// TIA Portal V16 export
// export: Created 2021-07-12T14:47:07.8764682Z, ExportSetting WithDefaults, DisplayName Totally Integrated Automation Portal, DisplayVersion V16, DisplayName TIA Portal Version Control Interface, DisplayVersion V16, DisplayName TIA Portal Openness, DisplayVersion V16, DisplayName STEP 7 Professional, DisplayVersion V16, DisplayName STEP 7 Safety, DisplayVersion V16, DisplayName WinCC Professional, DisplayVersion V16
FUNCTION_BLOCK "SimaHydTO_AxisAdvanced_PosAxis"   // FB33111, FBD
TITLE = SimaHydTO_AxisAdvanced_PosAxis
{ S7_Optimized_Access := 'TRUE' }
FAMILY : SimaHydTO/LAxisBasics
VERSION : 1.0
// Function block information: See Function block network 1
// stored: AutoNumber true, IsIECCheckEnabled false, IsRetainMemResEnabled false, MemoryReserve 100, SetENOAutomatically false, UDAEnableTagReadback false
   VAR_INPUT
      axis : TO_PositioningAxis;   // Technology object (axis)
      moveRelativeExecute : Bool;   // MC_MoveRelative: Start job with a positive edge
      moveRelativeDistance : LReal := 0.0;   // Distance of relative movement
      moveAbsoluteExecute : Bool;   // MC_MoveAbsolute: Start job with a positive edge
      moveAbsolutePosition : LReal := 0.0;   // Target position of absolute movement
      moveAbsoluteDirection : Int := 1;   // Direction of absolute movement: 0: Positive direction / 1: Negative direction / 3: Shortest direction
      moveAbsPositionControlled : Bool := true;   // 0: Non position-controlled operation / 1: Position-controlled mode - The parameter applies as long as the MC_MoveJog command is executed. After this, the setting of MC_Power applies again.
      haltExecute : Bool;   // MC_Halt: Start job with a positive edge
      haltAbortAcceleration : Bool := false;   // Acceleration control: False: The current acceleration at the start of the job is reduced using the configured jerk. Afterwards, the deceleration builds up / True: The acceleration is set to 0.0 at the start of the job, and the deceleration immediately builds up.
      Velocity : LReal := 100.0;   // Velocity of movement
      Acceleration : LReal := -1.0;   // Acceleration of movement
      Deceleration : LReal := -1.0;   // Deceleration of movement
      Jerk : LReal := -1.0;   // Jerk of movement
   END_VAR
   VAR_OUTPUT
      moveRelativeDone { ExternalWritable := 'False'} : Bool;   // MC_MoveRelative: Job is completed
      moveRelativeBusy { ExternalWritable := 'False'} : Bool;   // MC_MoveRelative: Job is running
      moveAbsoluteDone { ExternalWritable := 'False'} : Bool;   // MC_MoveAbsolute: Job is completed
      moveAbsoluteBusy { ExternalWritable := 'False'} : Bool;   // MC_MoveAbsolute: Job is running
      haltDone { ExternalWritable := 'False'} : Bool;   // MC_Halt: Job is running
      haltBusy { ExternalWritable := 'False'} : Bool;   // MC_Halt: Job is running
      commandAborted { ExternalWritable := 'False'} : Bool;   // The job was aborted by another job during execution (see also StatusID)
      error { ExternalWritable := 'False'} : Bool;   // An error occurred during execution of the job. The job is rejected. The cause of the error can be found in the "ErrorID" parameter.
      errorID { ExternalWritable := 'False'} : Word;   // ErrorID of motion control instruction (see also StatusID)
      statusID { ExternalWritable := 'False'} : Int;   // Additional specification of affected Motion control instruction of CommandAborted or Error: 0: No instruction / 1: MC_MoveRelative / 2: MC_MoveAbsolute / 3: MC_Halt
   END_VAR
   VAR
      instMcMoveRelative { ExternalAccessible := 'False'; ExternalVisible := 'False'; ExternalWritable := 'False'; S7_SetPoint := 'True'} : MC_MOVERELATIVE;   // PLCopen functions of basic motion control
      instMcMoveAbsolute { ExternalAccessible := 'False'; ExternalVisible := 'False'; ExternalWritable := 'False'; S7_SetPoint := 'True'} : MC_MOVEABSOLUTE;
      instMcHalt { ExternalAccessible := 'False'; ExternalVisible := 'False'; ExternalWritable := 'False'; S7_SetPoint := 'True'} : MC_HALT;
      statCommandAborted { ExternalAccessible := 'False'; ExternalVisible := 'False'; ExternalWritable := 'False'} : Array[#ARRAY_BEGIN..#ARRAY_END] of Bool;   // Arrays to save error information of PLCopen functions
      statError { ExternalAccessible := 'False'; ExternalVisible := 'False'; ExternalWritable := 'False'} : Array[#ARRAY_BEGIN..#ARRAY_END] of Bool;
      statErrorID { ExternalAccessible := 'False'; ExternalVisible := 'False'; ExternalWritable := 'False'} : Array[#ARRAY_BEGIN..#ARRAY_END] of Word;
      instMoveAbsOpenLoop { S7_SetPoint := 'True'} : "LSimaHydTO_MC_MoveAbsOpenLoop";
   END_VAR
   VAR_TEMP
      tempDwordCommandAborted : DWord;   // Variables to check error informations of PLCopen functions
      tempDwordError : DWord;
      tempCount : Int;   // Counter of FOR counting loop
   END_VAR
   VAR CONSTANT
      ARRAY_BEGIN : Int := 1;   // Start-Index of array (Maximum 32 Array elements!)
      ARRAY_END : Int := 32;   // End-Index of array (Maximum 32 Array elements!)
      ERROR_DEFAULT : Bool := false;   // Default values of output signals
      ERRORID_DEFAULT : Word := 16#0;
      STATUSID_DEFAULT : Int := 0;
   END_VAR
BEGIN

REGION Network 1 (SCL): Axis Basics - Header
   //=============================================================================
   //SIEMENS AG
   //(c)Copyright 2016 All Rights Reserved
   //-----------------------------------------------------------------------------
   //Library:       AxisAdvanced
   //Tested with:   S7-1500 V2.5
   //Engineering:   TIA Portal V15
   //Restrictions:  Motion Control Library V4.0
   //Requirements:  S7-1500(T)
   //Functionality: Advanced axis control of TO_PositioningAxis
   //-----------------------------------------------------------------------------
   //Change log table:
   //Version  Date       Expert in charge Changes applied
   //01.00.00 19.07.2019 ArSc             First released version
   //=============================================================================
END_REGION

REGION Network 2: Axis Advanced - MC_MoveRelative
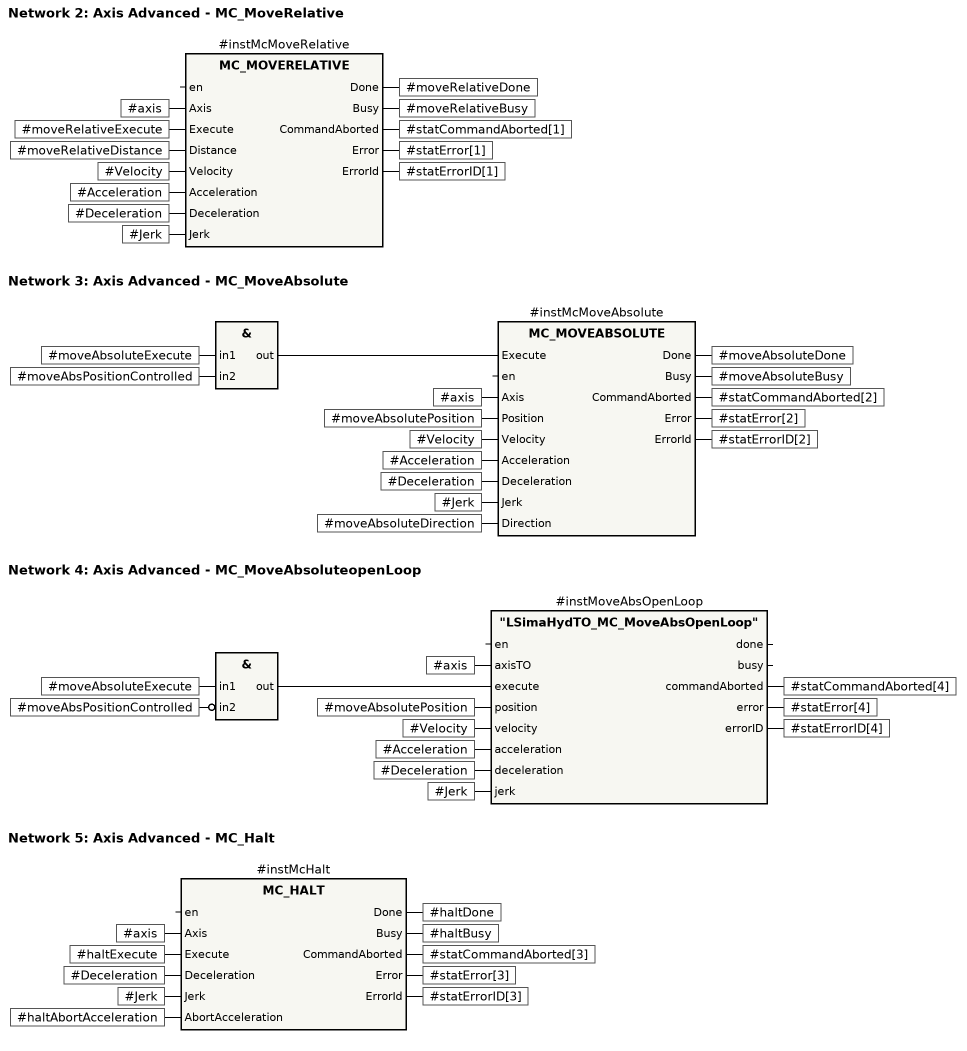
   #instMcMoveRelative(Axis := #axis,   // MC_MOVERELATIVE
                       Execute := #moveRelativeExecute,
                       Distance := #moveRelativeDistance,
                       Velocity := #Velocity,
                       Acceleration := #Acceleration,
                       Deceleration := #Deceleration,
                       Jerk := #Jerk,
                       Done => #moveRelativeDone,
                       Busy => #moveRelativeBusy,
                       CommandAborted => #statCommandAborted[1],
                       Error => #statError[1],
                       ErrorId => #statErrorID[1]);
END_REGION

REGION Network 3: Axis Advanced - MC_MoveAbsolute
   #instMcMoveAbsolute(Execute := #moveAbsoluteExecute AND #moveAbsPositionControlled,   // MC_MOVEABSOLUTE
                       Axis := #axis,
                       Position := #moveAbsolutePosition,
                       Velocity := #Velocity,
                       Acceleration := #Acceleration,
                       Deceleration := #Deceleration,
                       Jerk := #Jerk,
                       Direction := #moveAbsoluteDirection,
                       Done => #moveAbsoluteDone,
                       Busy => #moveAbsoluteBusy,
                       CommandAborted => #statCommandAborted[2],
                       Error => #statError[2],
                       ErrorId => #statErrorID[2]);
END_REGION

REGION Network 4: Axis Advanced - MC_MoveAbsoluteopenLoop
   #instMoveAbsOpenLoop(axisTO := #axis,   // "LSimaHydTO_MC_MoveAbsOpenLoop"
                        execute := #moveAbsoluteExecute AND NOT #moveAbsPositionControlled,
                        position := #moveAbsolutePosition,
                        velocity := #Velocity,
                        acceleration := #Acceleration,
                        deceleration := #Deceleration,
                        jerk := #Jerk,
                        commandAborted => #statCommandAborted[4],
                        error => #statError[4],
                        errorID => #statErrorID[4]);
END_REGION

REGION Network 5: Axis Advanced - MC_Halt
   #instMcHalt(Axis := #axis,   // MC_HALT
               Execute := #haltExecute,
               Deceleration := #Deceleration,
               Jerk := #Jerk,
               AbortAcceleration := #haltAbortAcceleration,
               Done => #haltDone,
               Busy => #haltBusy,
               CommandAborted => #statCommandAborted[3],
               Error => #statError[3],
               ErrorId => #statErrorID[3]);
END_REGION

REGION Network 6 (SCL): Axis Basics - Generate output signals and error detection
   //General output signals

   //Reset output signals
   #commandAborted := False;
   #error := False;
   #errorID := #ERRORID_DEFAULT;
   #statusID := #STATUSID_DEFAULT;

   //Transfer ARRAY to DWORD
   GATHER(IN:=#statCommandAborted,
          OUT=>#tempDwordCommandAborted);
   GATHER(IN:=#statError,
          OUT=>#tempDwordError);

   //Check for errors or command aborts
   IF (#tempDwordError > DWORD#0)
   THEN
     //Select error information
     FOR #tempCount := #ARRAY_BEGIN TO #ARRAY_END
     DO
       IF (#statError[#tempCount] = True)
       THEN
         #error := True;
         #errorID := #statErrorID[#tempCount];
         #statusID := #tempCount;
         EXIT;
       END_IF;
     END_FOR;
   ELSIF (#tempDwordCommandAborted > DWORD#0)
   THEN
     //Select command aborted information
     FOR #tempCount := #ARRAY_BEGIN TO #ARRAY_END
     DO
       IF (#statCommandAborted[#tempCount] = True)
       THEN
         #commandAborted := True;
         #errorID := #statErrorID[#tempCount];
         #statusID := #tempCount;
         EXIT;
       END_IF;
     END_FOR;
   END_IF;
END_REGION
END_FUNCTION_BLOCK
